TYPE ST_IvekCommandBits :
STRUCT
	// TODO: Confirm bit positions against the EDS/manual matching installed firmware.
    nDispenseBit         : USINT := 0;
    nStopBit             : USINT := 1;
    nClearFaultBit       : USINT := 2;
    nReferenceBit        : USINT := 3;
END_STRUCT
END_TYPE

(* stored: Version 1.1.0.1, ProductVersion 3.1.4026.18
   DUT ST_IvekCommandBits: Id {f78fb8cb-ad64-4e90-bf6e-f4552c1d9bc4} *)
